(* IEC 61131-3 sources: Lasal/CPU_5344_V01/Class/cntrAmount, 1 file *)

(* ---- cntrAmount.st ---- *)
(*!
<Class
	Name               = "cntrAmount"
	Revision           = "0.0"
	RealtimeTask       = "false"
	CyclicTask         = "false"
	BackgroundTask     = "true"
	DefBackground      = "100 ms"
	Sigmatek           = "false"
	OSInterface        = "false"
	HighPriority       = "false"
	Automatic          = "false"
	UpdateMode         = "Prescan"
	SharedCommandTable = "true"
	Objectsize         = "(284,120)">
	<Channels>
		<Server Name="ClassSvr" Visualized="false" Initialize="false" WriteProtected="true" Retentive="false"/>
		<Server Name="count" Visualized="false" Initialize="false" WriteProtected="false" Retentive="false"/>
		<Server Name="resetSoftCounter" Visualized="true" Initialize="false" WriteProtected="false" Retentive="false"/>
		<Server Name="softCounter" Visualized="true" Initialize="false" WriteProtected="false" Retentive="SRam"/>
		<Server Name="totalCounter" Visualized="true" Initialize="false" WriteProtected="false" Retentive="SRam"/>
	</Channels>
</Class>
*)
cntrAmount : CLASS
  //Servers:
	ClassSvr 	: SvrChCmd_DINT;
	softCounter 	: SvrCh_DINT;
	totalCounter 	: SvrCh_DINT;
	resetSoftCounter 	: SvrCh_DINT;
	count 	: SvrCh_DINT;
  //Clients:
  //Variables:
		tmpCounter 	: DINT;
		timeWritten 	: UDINT;
  //Functions:

	FUNCTION VIRTUAL GLOBAL Init;

	FUNCTION VIRTUAL GLOBAL Background
		VAR_INPUT
			EAX 	: UDINT;
		END_VAR
		VAR_OUTPUT
			state (EAX) 	: UDINT := READY;
		END_VAR;

	FUNCTION storeIt;

	FUNCTION VIRTUAL GLOBAL resetSoftCounter::Write
		VAR_INPUT
			input (EAX) 	: DINT;
		END_VAR
		VAR_OUTPUT
			result (EAX) 	: DINT;
		END_VAR;

	FUNCTION VIRTUAL GLOBAL count::Write
		VAR_INPUT
			input (EAX) 	: DINT;
		END_VAR
		VAR_OUTPUT
			result (EAX) 	: DINT;
		END_VAR;
  //Tables:
	FUNCTION @STD
		VAR_OUTPUT
			ret_code	: CONFSTATES;
		END_VAR;
	FUNCTION GLOBAL TAB @CT_;
END_CLASS;

// JdK 21-11-2019: class to count operations, they are stored in ram servers, don't write them to often

FUNCTION VIRTUAL GLOBAL cntrAmount::Init

  tmpCounter:= totalCounter;
  timeWritten:= ops.tAbsolute;

END_FUNCTION

FUNCTION VIRTUAL GLOBAL cntrAmount::Background
	VAR_INPUT
		EAX 	: UDINT;
	END_VAR
	VAR_OUTPUT
		state (EAX) 	: UDINT;(* := READY *)
	END_VAR

  IF totalCounter= tmpCounter THEN
    timeWritten:= ops.tAbsolute; //no need to write again
  ELSIF ops.tAbsolute-timeWritten > 300000 THEN //after 5 minutes
    storeIt();
  END_IF;

END_FUNCTION

FUNCTION VIRTUAL GLOBAL cntrAmount::resetSoftCounter::Write
	VAR_INPUT
		input (EAX) 	: DINT;
	END_VAR
	VAR_OUTPUT
		result (EAX) 	: DINT;
	END_VAR

	resetSoftCounter := input;
  softCounter:= 0;
  softCounter.Write(input:=softCounter);
	result := resetSoftCounter;

END_FUNCTION

FUNCTION VIRTUAL GLOBAL cntrAmount::count::Write
	VAR_INPUT
		input (EAX) 	: DINT;
	END_VAR
	VAR_OUTPUT
		result (EAX) 	: DINT;
	END_VAR

	count := input;

  softCounter+=1;
  totalCounter+=1;

  IF totalCounter - tmpCounter > 100 THEN //don't write every action, to safe memory
    storeIt();
  END_IF;

	result := count;

END_FUNCTION

FUNCTION cntrAmount::storeIt

  tmpCounter:=totalCounter;
  softCounter-= 1; //we can only store a new value
  totalCounter-= 1;
  softCounter.Write(input:=softCounter+1); //write action to store value
  totalCounter.Write(input:=totalCounter+1);

END_FUNCTION
